# EPICS substitutions: iocbio4/iocBoot/UNUSED/canberra_13.substitutions
file "$(MCA)/mcaApp/Db/simple_mca.db"
{
pattern
{P           M       DTYP           INP         PREC  CHANS}
{18IDd:med:   mca1  "asynMCA"   "@asyn(AIM2/1 0)"    3  2048}
{18IDd:med:   mca2  "asynMCA"   "@asyn(AIM2/1 1)"    3  2048}
{18IDd:med:   mca3  "asynMCA"   "@asyn(AIM2/1 2)"    3  2048}
{18IDd:med:   mca4  "asynMCA"   "@asyn(AIM2/2 0)"    3  2048}
{18IDd:med:   mca5  "asynMCA"   "@asyn(AIM2/2 1)"    3  2048}
{18IDd:med:   mca6  "asynMCA"   "@asyn(AIM2/2 2)"    3  2048}
{18IDd:med:   mca7  "asynMCA"   "@asyn(AIM3/1 0)"    3  2048}
{18IDd:med:   mca8  "asynMCA"   "@asyn(AIM3/1 1)"    3  2048}
{18IDd:med:   mca9  "asynMCA"   "@asyn(AIM3/1 2)"    3  2048}
{18IDd:med:   mca10 "asynMCA"   "@asyn(AIM3/2 0)"    3  2048}
{18IDd:med:   mca11 "asynMCA"   "@asyn(AIM3/3 1)"    3  2048}
{18IDd:med:   mca12 "asynMCA"   "@asyn(AIM3/4 2)"    3  2048}
{18IDd:med:   mca13 "asynMCA"   "@asyn(AIM3/2 3)"    3  2048}
{18IDd:med:   mca0  "Soft Channel"   ""     3  2048}
}

file "$(MCA)/mcaApp/Db/icb_amp.db"
{
pattern
{P			AMP		PORT}
{18IDd:med:	amp1	"icbAmp1"}
{18IDd:med:	amp2	"icbAmp2"}
{18IDd:med:	amp3	"icbAmp3"}
{18IDd:med:	amp4	"icbAmp4"}
{18IDd:med:	amp5	"icbAmp5"}
{18IDd:med:	amp6	"icbAmp6"}
{18IDd:med:	amp7	"icbAmp7"}
{18IDd:med:	amp8	"icbAmp8"}
{18IDd:med:	amp9	"icbAmp9"}
{18IDd:med:	amp10	"icbAmp10"}
{18IDd:med:	amp11	"icbAmp11"}
{18IDd:med:	amp12	"icbAmp12"}
{18IDd:med:	amp13	"icbAmp13"}
}

file "$(MCA)/mcaApp/Db/icb_adc.db"
{
pattern
{P			ADC		PORT}
{18IDd:med:	adc1	"icbAdc1"}
{18IDd:med:	adc2	"icbAdc2"}
{18IDd:med:	adc3	"icbAdc3"}
{18IDd:med:	adc4	"icbAdc4"}
}

file "$(MCA)/mcaApp/Db/icb_hvps.db"
{
pattern
{P			HVPS	LIMIT	PORT}
{18IDd:med:	hvps1	1000	"icbHvps1"}
}
